// TIA Portal V17 export
// export: Created 2024-09-03T21:54:57.8014129Z, ExportSetting WithDefaults, DisplayName Totally Integrated Automation Portal, DisplayVersion V17 Update 7, DisplayName TIA Portal Openness, DisplayVersion V17 Update 7, DisplayName TIA Portal Version Control Interface, DisplayVersion V17, DisplayName SINAMICS Startdrive Advanced, DisplayVersion V17 SP2, DisplayName SINAMICS Startdrive G110M, G120, G120C, G120D, G120P, G115D, DisplayVersion V17 SP2, DisplayName SINAMICS Startdrive G130, G150, S120, S150, SINAMICS MV, S210, DisplayVersion V17 SP2, DisplayName STEP 7 Professional, DisplayVersion V17 Update 7, DisplayName STEP 7 Safety, DisplayVersion V17 Update 6, DisplayName WinCC Advanced / Unified PC, DisplayVersion V17 Update 7
DATA_BLOCK "SystemHMI"   // DB10
{ S7_Optimized_Access := 'TRUE' }
VERSION : 0.1
// stored: AutoNumber false, DBAccessibleFromOPCUA true, DBAccessibleFromWebserver true, IsOnlyStoredInLoadMemory false, IsRetainMemResEnabled false, IsWriteProtectedInAS false, MemoryReserve 100
   VAR
      AlarmActive : Bool := FALSE;
      AlarmActiveBlinking : Bool := FALSE;
      WarningActive : Bool := FALSE;
      BasicPosition : Bool := FALSE;
      GoToBasicPosition : Bool := FALSE;
      ManualMode : Bool := TRUE;
      AutomaticMode : Bool := FALSE;
      ManualCommand : Int := 0;
      BasicPositionMessage : Int := 0;
      BasicPositionStep : Int := 0;
      ManualFromRobot : Bool := FALSE;
      HydraulicPumpAutoControl : Bool := FALSE;
      BasicPositionSt1 : Bool := FALSE;
      BasicPositionSt2 : Bool := FALSE;
      BasicPositionFitting : Bool := FALSE;
      BasicPositionGripper1 : Bool := FALSE;
      BasicPositionStartHMI : Bool := FALSE;
      AutoStartHMI : Bool := FALSE;
      ResetPartsErrors : Bool := FALSE;
      ModeChanged : Bool := FALSE;
   END_VAR
BEGIN
END_DATA_BLOCK
